// TIA Portal project "Sortier_Station_0" (V20)

(* hardware
DEVICE "S7-1500/ET200MP-Station_1"  S7-1500 station
   slot 0: "Profilschiene_0"  Rack  6ES7 590-1***0-0AA0
   slot 1: "PLC_1"  CPU 1513-1 PN  6ES7 513-1AM03-0AB0  V4.0
      slot 3: "CPU-Display_1"  6ES7591-1AA00-0AA0
      slot 32768: "PROFINET-Schnittstelle_1"  X1
         slot 32769: "Port_1"  X1 P1
         slot 32770: "Port_2"  X1 P2
      slot 34817: "Virtual CP interface port_1"  Virtual CP interface port  Virtual CP interface port FW V4.0
   slot 2: "DI 16x24VDC BA_1"  DI 16x24VDC BA  6ES7 521-1BH10-0AA0  V1.1
   slot 3: "DQ 16x24VDC/0.5A ST_1"  DQ 16x24VDC/0.5A ST  6ES7 522-1BH00-0AB0  V2.0
   slot 4: "AI 8xU/I/R/RTD BA_1"  AI 8xU/I/R/RTD BA  6ES7 531-7QF00-0AB0  V1.0
   slot 5: "AQ 8xU/I HS_1"  AQ 8xU/I HS  6ES7 532-5HF00-0AB0  V2.2
   slot 6: "AI 8xU/I/R/RTD BA_2"  AI 8xU/I/R/RTD BA  6ES7 531-7QF00-0AB0  V1.0
   slot 7: "AQ 8xU/I HS_2"  AQ 8xU/I HS  6ES7 532-5HF00-0AB0  V2.2
*)

// ===== PLC "PLC_1"  CPU 1513-1 PN =====

VAR_GLOBAL   // PLC tag table "Standard-Variablentabelle"
   "PlcLabConnectIn01" AT %ID32760 : DWord;
   "PlcLabConnectIn02" AT %ID32764 : DWord;
   "PlcLabConnectOut01" AT %QD32760 : DWord;
   "PlcLabConnectOut02" AT %QD32764 : DWord;
   "Clock_Byte" AT %MB0 : Byte;
   "Clock_10Hz" AT %M0.0 : Bool;
   "Clock_5Hz" AT %M0.1 : Bool;
   "Clock_2.5Hz" AT %M0.2 : Bool;
   "Clock_2Hz" AT %M0.3 : Bool;
   "Clock_1.25Hz" AT %M0.4 : Bool;
   "Clock_1Hz" AT %M0.5 : Bool;
   "Clock_0.625Hz" AT %M0.6 : Bool;
   "Clock_0.5Hz" AT %M0.7 : Bool;
END_VAR

VAR_GLOBAL   // PLC tag table "Eingaenge"
   "S1" AT %I0.0 : Bool;   // Not-Aus Schalter
   "S2" AT %I0.1 : Bool;   // Betriebsschalter
   "S3" AT %I0.2 : Bool;   // Starttaster
   "S4" AT %I0.3 : Bool;   // Stopptaster
   "S5" AT %I0.4 : Bool;   // Resettaster
   "2b1" AT %I1.0 : Bool;   // Lichtschranke am Ausgang (Reflektor)
   "1b1" AT %ID30 : DInt;   // Visionsensor am Eingang
END_VAR

VAR_GLOBAL   // PLC tag table "Ausgaenge"
   "H1" AT %Q0.2 : Bool;   // Startleuchte
   "H2" AT %Q0.3 : Bool;   // Stoppleuchte
   "H3" AT %Q0.4 : Bool;   // Resetleuchte
   "M1" AT %A0.5 : Bool;   // Zulauf Förderband
   "M2" AT %A0.6 : Bool;   // Auslauf Förderband
   "M3" AT %A0.7 : Bool;   // Stopp-Barriere
   "1M1" AT %Q1.3 : Bool;   // Sortierer (rechts)
   "2M1" AT %Q1.4 : Bool;   // Sortierer (mittig)
   "3M1" AT %Q1.5 : Bool;   // Sortierer (links)
   "D1" AT %QD30 : DInt;   // Zähleranzeige (rechts)
   "D2" AT %QD34 : DInt;   // Zähleranzeige (mittig)
   "D3" AT %QD38 : DInt;   // Zähleranzeige (links)
   "1M2" AT %A1.0 : Bool;   // Sortiererband (rechts)
   "2M2" AT %A1.1 : Bool;   // Sortiererband (mittig)
   "3M2" AT %A1.2 : Bool;   // Sortiererband (links)
END_VAR

DATA_BLOCK "Sortierdaten"   // DB2
{ S7_Optimized_Access := 'TRUE' }
VERSION : 0.1
   VAR
      Anlagendaten : Struct
         NotAus_aktiv : Bool;
         Anlage_aktiv : Bool;
      END_STRUCT;
      Bauteil : Struct
         Blau : Bool;
         Gruen : Bool;
         Grau : Bool;
      END_STRUCT;
      Betriebsdaten : Struct
         Blaues_Teil_erkannt : Bool;   // Blaues Teil in Anlage
         Gruenes_Teil_erkannt : Bool;   // Grünes Teil in Anlage
         Graues_Teil_erkannt : Bool;   // Graues Teil in Anlage
         PTRIG_2b1 : Bool;
         Teil_in_Auslass : Bool;   // Bauteil hat die Anlage verlassen
         Teil_in_Einlass : Bool;
         Einlass_aktiv : Bool;
         Barriere_aktiv : Bool;
         Sortierermotoren : Struct
            "1M1" : Bool;
            "2M1" : Bool;
            "3M1" : Bool;
         END_STRUCT;
      END_STRUCT;
   END_VAR
   VAR RETAIN
      Zaehler : Struct   // Zum speichern der Zähler der Bauteile im Auslauf Förderband
         Blau : DInt;
         Gruen : DInt;
         Grau : DInt;
      END_STRUCT;
   END_VAR
BEGIN
END_DATA_BLOCK

// folder: System blocks/Program resources

DATA_BLOCK "IEC_Counter_0_DB"   // DB1
{ S7_Optimized_Access := 'TRUE' }
AUTHOR : SIMATIC
FAMILY : IEC
NAME : DCNTR
VERSION : 1.2
// stored: InstanceOfName IEC_DCOUNTER
"IEC_DCOUNTER"
BEGIN
END_DATA_BLOCK

DATA_BLOCK "IEC_Counter_0_DB_1"   // DB3
{ S7_Optimized_Access := 'TRUE' }
AUTHOR : SIMATIC
FAMILY : IEC
NAME : DCNTR
VERSION : 1.2
// stored: InstanceOfName IEC_DCOUNTER
"IEC_DCOUNTER"
BEGIN
END_DATA_BLOCK

DATA_BLOCK "IEC_Counter_0_DB_2"   // DB4
{ S7_Optimized_Access := 'TRUE' }
AUTHOR : SIMATIC
FAMILY : IEC
NAME : DCNTR
VERSION : 1.2
// stored: InstanceOfName IEC_DCOUNTER
"IEC_DCOUNTER"
BEGIN
END_DATA_BLOCK

DATA_BLOCK "IEC_Timer_0_DB"   // DB5
{ S7_Optimized_Access := 'TRUE' }
AUTHOR : Simatic
FAMILY : IEC
NAME : IEC_TMR
VERSION : 1.0
// stored: InstanceOfName IEC_TIMER
"IEC_TIMER"
BEGIN
END_DATA_BLOCK

DATA_BLOCK "IEC_Counter_0_DB_5"   // DB7
{ S7_Optimized_Access := 'TRUE' }
AUTHOR : Simatic
FAMILY : IEC
NAME : CNTR
VERSION : 1.0
// stored: InstanceOfName IEC_COUNTER
"IEC_COUNTER"
BEGIN
END_DATA_BLOCK

// folder: (top level)

FUNCTION "Bandsteuerung" : Void   // FC1, FBD
{ S7_Optimized_Access := 'TRUE' }
VERSION : 0.1
   VAR_TEMP   // added for the SCL form of the ladder/FBD networks
      _w1 : Bool;
      _w2 : Bool;
   END_VAR
BEGIN

REGION Network 1: Anlagensteuerung
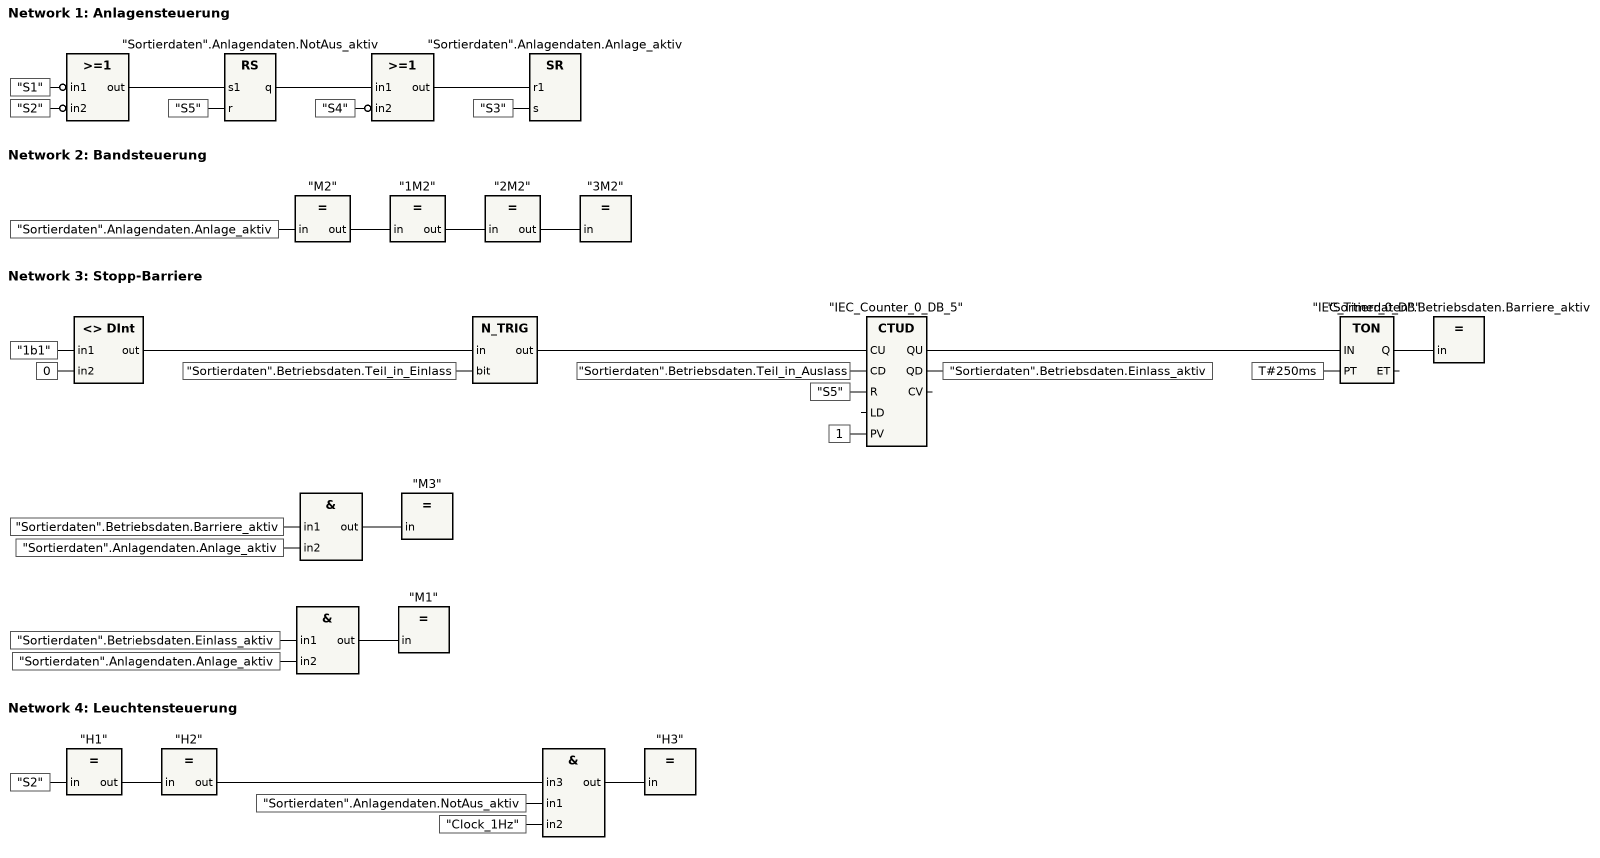
   IF "S5" THEN
       "Sortierdaten".Anlagendaten.NotAus_aktiv := FALSE;   // RS flip-flop
   END_IF;
   IF NOT "S1" OR NOT "S2" THEN "Sortierdaten".Anlagendaten.NotAus_aktiv := TRUE; END_IF;
   IF "S3" THEN
       "Sortierdaten".Anlagendaten.Anlage_aktiv := TRUE;   // SR flip-flop
   END_IF;
   IF "Sortierdaten".Anlagendaten.NotAus_aktiv OR NOT "S4" THEN
       "Sortierdaten".Anlagendaten.Anlage_aktiv := FALSE;
   END_IF;
END_REGION

REGION Network 2: Bandsteuerung
   "M2" := "Sortierdaten".Anlagendaten.Anlage_aktiv;
   "1M2" := "Sortierdaten".Anlagendaten.Anlage_aktiv;
   "2M2" := "Sortierdaten".Anlagendaten.Anlage_aktiv;
   "3M2" := "Sortierdaten".Anlagendaten.Anlage_aktiv;
END_REGION

REGION Network 3: Stopp-Barriere
   #_w1 := "1b1" <> 0;
   #_w2 := NOT #_w1 AND "Sortierdaten".Betriebsdaten.Teil_in_Einlass;   // falling edge
   "Sortierdaten".Betriebsdaten.Teil_in_Einlass := #_w1;
   "IEC_Counter_0_DB_5".CTUD(CU := #_w2,
                           CD := "Sortierdaten".Betriebsdaten.Teil_in_Auslass,
                           R := "S5",
                           PV := 1,
                           QD => "Sortierdaten".Betriebsdaten.Einlass_aktiv);
   "IEC_Timer_0_DB".TON(IN := "IEC_Counter_0_DB_5".QU, PT := T#250ms);
   "Sortierdaten".Betriebsdaten.Barriere_aktiv := "IEC_Timer_0_DB".Q;
   "M3" := "Sortierdaten".Betriebsdaten.Barriere_aktiv AND "Sortierdaten".Anlagendaten.Anlage_aktiv;
   "M1" := "Sortierdaten".Betriebsdaten.Einlass_aktiv AND "Sortierdaten".Anlagendaten.Anlage_aktiv;
END_REGION

REGION Network 4: Leuchtensteuerung
   "H1" := "S2";
   "H2" := "S2";
   "H3" := "S2" AND "Sortierdaten".Anlagendaten.NotAus_aktiv AND "Clock_1Hz";
END_REGION
END_FUNCTION

FUNCTION "Sortiersteuerung" : Void   // FC2, FBD
{ S7_Optimized_Access := 'TRUE' }
VERSION : 0.1
   VAR_TEMP   // added for the SCL form of the ladder/FBD networks
      _w1 : Bool;
      _w2 : Bool;
   END_VAR
BEGIN

REGION Network 1: Sortierer (rechts)
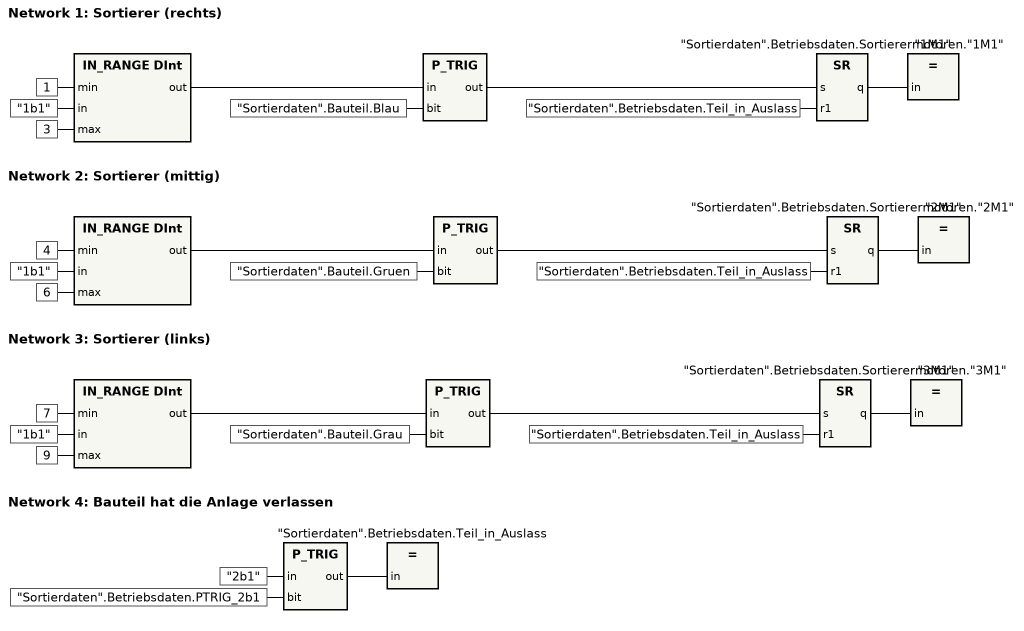
   #_w1 := (1 <= "1b1") AND ("1b1" <= 3);
   #_w2 := #_w1 AND NOT "Sortierdaten".Bauteil.Blau;   // rising edge
   "Sortierdaten".Bauteil.Blau := #_w1;
   IF #_w2 THEN
       "Sortierdaten".Betriebsdaten.Sortierermotoren."1M1" := TRUE;   // SR flip-flop
   END_IF;
   IF "Sortierdaten".Betriebsdaten.Teil_in_Auslass THEN
       "Sortierdaten".Betriebsdaten.Sortierermotoren."1M1" := FALSE;
   END_IF;
   "1M1" := "Sortierdaten".Betriebsdaten.Sortierermotoren."1M1";
END_REGION

REGION Network 2: Sortierer (mittig)
   #_w1 := (4 <= "1b1") AND ("1b1" <= 6);
   #_w2 := #_w1 AND NOT "Sortierdaten".Bauteil.Gruen;   // rising edge
   "Sortierdaten".Bauteil.Gruen := #_w1;
   IF #_w2 THEN
       "Sortierdaten".Betriebsdaten.Sortierermotoren."2M1" := TRUE;   // SR flip-flop
   END_IF;
   IF "Sortierdaten".Betriebsdaten.Teil_in_Auslass THEN
       "Sortierdaten".Betriebsdaten.Sortierermotoren."2M1" := FALSE;
   END_IF;
   "2M1" := "Sortierdaten".Betriebsdaten.Sortierermotoren."2M1";
END_REGION

REGION Network 3: Sortierer (links)
   #_w1 := (7 <= "1b1") AND ("1b1" <= 9);
   #_w2 := #_w1 AND NOT "Sortierdaten".Bauteil.Grau;   // rising edge
   "Sortierdaten".Bauteil.Grau := #_w1;
   IF #_w2 THEN
       "Sortierdaten".Betriebsdaten.Sortierermotoren."3M1" := TRUE;   // SR flip-flop
   END_IF;
   IF "Sortierdaten".Betriebsdaten.Teil_in_Auslass THEN
       "Sortierdaten".Betriebsdaten.Sortierermotoren."3M1" := FALSE;
   END_IF;
   "3M1" := "Sortierdaten".Betriebsdaten.Sortierermotoren."3M1";
END_REGION

REGION Network 4: Bauteil hat die Anlage verlassen
   #_w1 := "2b1" AND NOT "Sortierdaten".Betriebsdaten.PTRIG_2b1;   // rising edge
   "Sortierdaten".Betriebsdaten.PTRIG_2b1 := "2b1";
   "Sortierdaten".Betriebsdaten.Teil_in_Auslass := #_w1;
END_REGION
END_FUNCTION

FUNCTION "Zaehlersteuerung" : Void   // FC3, FBD
{ S7_Optimized_Access := 'TRUE' }
VERSION : 0.1
BEGIN

REGION Network 1: Zähler (blaue Teile)
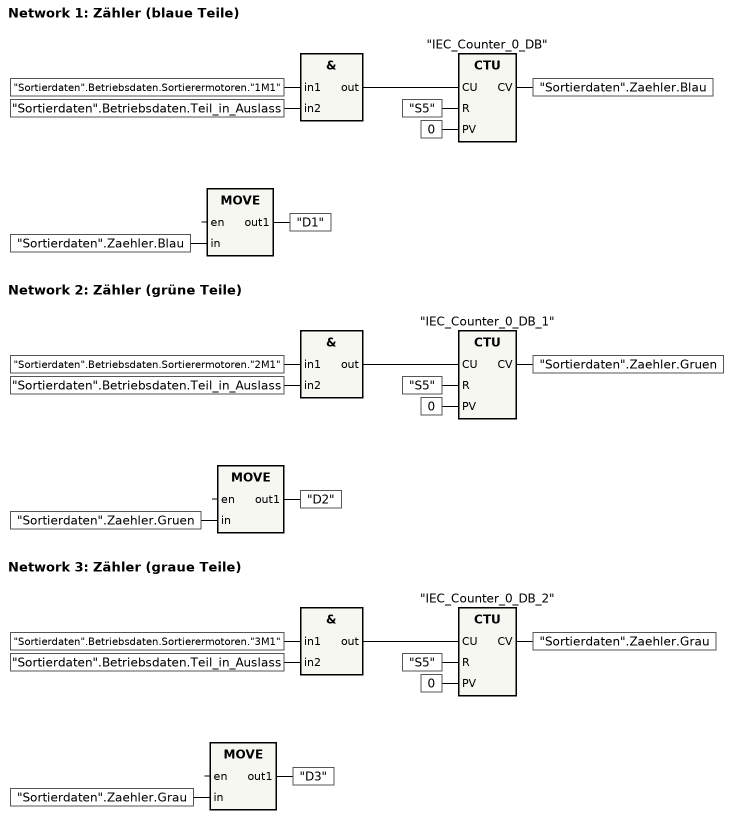
   "IEC_Counter_0_DB".CTU(CU := "Sortierdaten".Betriebsdaten.Sortierermotoren."1M1" AND "Sortierdaten".Betriebsdaten.Teil_in_Auslass,
                          R := "S5",
                          PV := 0,
                          CV => "Sortierdaten".Zaehler.Blau);
   "D1" := "Sortierdaten".Zaehler.Blau;
END_REGION

REGION Network 2: Zähler (grüne Teile)
   "IEC_Counter_0_DB_1".CTU(CU := "Sortierdaten".Betriebsdaten.Sortierermotoren."2M1" AND "Sortierdaten".Betriebsdaten.Teil_in_Auslass,
                           R := "S5",
                           PV := 0,
                           CV => "Sortierdaten".Zaehler.Gruen);
   "D2" := "Sortierdaten".Zaehler.Gruen;
END_REGION

REGION Network 3: Zähler (graue Teile)
   "IEC_Counter_0_DB_2".CTU(CU := "Sortierdaten".Betriebsdaten.Sortierermotoren."3M1" AND "Sortierdaten".Betriebsdaten.Teil_in_Auslass,
                           R := "S5",
                           PV := 0,
                           CV => "Sortierdaten".Zaehler.Grau);
   "D3" := "Sortierdaten".Zaehler.Grau;
END_REGION
END_FUNCTION

ORGANIZATION_BLOCK "Main"   // OB1, FBD, ProgramCycle
TITLE = "Main Program Sweep (Cycle)"
{ S7_Optimized_Access := 'TRUE' }
VERSION : 0.1
   VAR_INPUT
      Initial_Call : Bool;   // Initial call of this OB
      Remanence : Bool;   // =True, if remanent data are available
   END_VAR
BEGIN

REGION Network 1
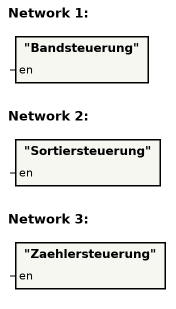
   "Bandsteuerung"();
END_REGION

REGION Network 2
   "Sortiersteuerung"();
END_REGION

REGION Network 3
   "Zaehlersteuerung"();
END_REGION
END_ORGANIZATION_BLOCK